// TIA Portal V17 export
// export: Created 2023-02-13T11:16:11.9834469Z, ExportSetting WithDefaults, DisplayName Totally Integrated Automation Portal, DisplayVersion V17, DisplayName TIA Portal Openness, DisplayVersion V17, DisplayName TIA Portal Teamcenter Gateway, DisplayVersion V17, DisplayName TIA Portal Version Control Interface, DisplayVersion V17, DisplayName SINAMICS Startdrive Advanced, DisplayVersion V17, DisplayName SINAMICS Startdrive G130, G150, S120, S150, SINAMICS MV, S210, DisplayVersion V17, DisplayName SINAMICS Startdrive G110M, G120, G120C, G120D, G120P, G115D, DisplayVersion V17, DisplayName STEP 7 Professional, DisplayVersion V17, DisplayName STEP 7 Safety, DisplayVersion V17, DisplayName WinCC Professional, DisplayVersion V17
DATA_BLOCK "General_Blend"   // DB33
{ S7_Optimized_Access := 'TRUE' }
VERSION : 0.1
// stored: AutoNumber true, DBAccessibleFromOPCUA true, DBAccessibleFromWebserver true, IsOnlyStoredInLoadMemory false, IsRetainMemResEnabled false, IsWriteProtectedInAS false, MemoryReserve 100
   VAR
      Drain_ON_OFF_THE1 : Bool;
      Drain_ON_OFF_THE2 : Bool;
      Blend_Cluster1 : Struct
         CIP_Line1 : Struct
            "CIP Enable" : Bool;
            "CIP Request" : Bool;
            V_Cmd : Bool;
            P_Cmd : Bool;
            P_SP : Real;
         END_STRUCT;
         CIP_Line2 : Struct
            "CIP Enable" : Bool;
            "CIP Request" : Bool;
            V_Cmd : Bool;
            P_Cmd : Bool;
            P_SP : Real;
         END_STRUCT;
         CIP_Line3 : Struct
            "CIP Enable" : Bool;
            "CIP Request" : Bool;
            V_Cmd : Bool;
            P_Cmd : Bool;
            P_SP : Real;
         END_STRUCT;
         ptrig : Bool;
      END_STRUCT;
      Blend_Cluster2 : Struct
         CIP_Line1 : Struct
            "CIP Enable" : Bool;
            "CIP Request" : Bool;
            V_Cmd : Bool;
            P_Cmd : Bool;
            P_SP : Real;
         END_STRUCT;
         CIP_Line2 : Struct
            "CIP Enable" : Bool;
            "CIP Request" : Bool;
            V_Cmd : Bool;
            P_Cmd : Bool;
            P_SP : Real;
         END_STRUCT;
         CIP_Line3 : Struct
            "CIP Enable" : Bool;
            "CIP Request" : Bool;
            V_Cmd : Bool;
            P_Cmd : Bool;
            P_SP : Real;
         END_STRUCT;
         ptrig : Bool;
      END_STRUCT;
      CIP_Bypass : Bool;
      "THE-4" : Struct
         "Timer" : TON_TIME;
         MSec { S7_SetPoint := 'True'} : DInt;
         Sec : DInt := 10;
         Act : DInt;
      END_STRUCT;
      "THE-5" : Struct
         "Timer" : TON_TIME;
         MSec { S7_SetPoint := 'True'} : DInt;
         Sec : DInt := 10;
         Act : DInt;
      END_STRUCT;
      Sugar : Struct
         "In Process" : Struct
            "T-20" : Bool;
            "T-21" : Bool;
            "T-30" : Bool;
            "T-31" : Bool;
            "T-40" : Bool;
            "T-41" : Bool;
         END_STRUCT;
      END_STRUCT;
   END_VAR
BEGIN
END_DATA_BLOCK
